(*********************************** G.D S.p.A. - Technical Department ***********************************
============= PROGRAM INFO ============
FOLDER:             TBD
MACHINES INVOLVED:  TBD 

============= DESCRIPTION =============
csp machine declaration

============= REVISIONS ===============
Date		Version	 	Author      	Description             
----------	-------		------------  	--------------------------------------------
2019/04/05 	0000.00	 	M.Grasso		Creation of the PRG

**********************************************************************************************************)
(*$R process_ref := prc; $*)
PROGRAM csp_transfer_accumulator_accU
VAR
	
	prc:											process;
	prc_path:										STRING;
	
END_VAR

_read_var_input();

_object_manager();

IF NOT objects_running()
THEN
	RETURN;	
END_IF

_read_process_image();

_mode_manager();

_set_runtime_properties();

(********************************* BODY *********************************)
(************************************************************************)

_handle_messages();

_write_output();

ACTION _handle_messages:
;
END_ACTION

ACTION _handle_process_test:
;
END_ACTION

ACTION _mode_manager:
IF process_mode_req_is_pending(prc)
THEN
    process_apply_mode_req_first_step(prc);
    CASE process_get_mode(prc) OF
        MODE_TO_ABSENT:
			;
        MODE_TO_INACTIVE:
			;
        MODE_TO_TEST:
			;
        MODE_TO_OPERATIONAL:
			;
    END_CASE
    process_apply_mode_req_second_step(prc);
END_IF
END_ACTION

ACTION _object_manager:
IF objects_initialization()
THEN
	sub_process_init(
		object_name					:= 'csp_transfer_accumulator_accU.prc', 
		process						:= csp_transfer_accumulator.prc, 
		CONVERSION_this				:= prc);
		
	prc_path 						:= process_get_path(prc);
END_IF

IF objects_running()
THEN
	process_cycle(prc);
END_IF
END_ACTION

ACTION _read_process_image:
;
END_ACTION

ACTION _read_var_input:
;
END_ACTION

ACTION _set_runtime_properties:
;
END_ACTION

ACTION _write_output:
;
END_ACTION

END_PROGRAM

(* stored: Version 1.1.0.1, ProductVersion 3.1.4022.12
   POU csp_transfer_accumulator_accU: Id {5a18f031-6baf-49aa-aa7d-093e662cf16b}, SpecialFunc None
   Action _handle_messages: Id {209b258f-5a54-4d2e-afc2-700c4a727a0e}
   Action _handle_process_test: Id {84aa30d9-3074-4463-b0db-363c02b6d16e}
   Action _mode_manager: Id {4f81e869-9d34-40e8-8f9b-9fd95459f84b}
   Action _object_manager: Id {af9411a1-ca1b-48e7-b2af-734c74af0436}
   Action _read_process_image: Id {a21635a2-4bd5-4f81-bc24-5f2c0d901d94}
   Action _read_var_input: Id {6efe5fc2-a9c8-44ac-93fc-de5625690d29}
   Action _set_runtime_properties: Id {0233ea32-5c4d-4776-ab9d-26ef00510775}
   Action _write_output: Id {e2c429bd-e239-4652-9b2c-9127d5fee7a8} *)
